FUNCTION WRITE_ANY_BOOL : BOOL
VAR_INPUT
    ptr: POINTER TO BOOL;
    val: BOOL;
END_VAR

ptr^ := val;

END_FUNCTION

(* stored: Version 1.1.0.1, ProductVersion 3.1.4022.9
   POU WRITE_ANY_BOOL: Id {d1649341-8878-4827-b4ef-c286e7025184}, SpecialFunc None *)
